TYPE I8 : SINT; END_TYPE

(* stored: Version 1.1.0.1
   DUT I8: Id {86095448-a507-0b1d-3eb9-ba8333db0b2e} *)
